PROGRAM MAIN
VAR
	nCounter	:DINT;
END_VAR

nCounter:=nCounter+1;

END_PROGRAM

(* stored: Version 1.1.0.1
   POU MAIN: Id {5554568d-2c6c-48fe-984c-7179df35e35b}, SpecialFunc None *)
